TYPE ST_SafetyDoor_IN :
STRUCT
	bStartButton : BOOL;
	bRequestButton : BOOL;
	bLockButton : BOOL;
	bLocked : BOOL;
	tsSafe : BOOL;
	tsOpen : BOOL;
	tsSegment_Open : BOOL;
END_STRUCT
END_TYPE

(* stored: Version 1.1.0.1
   DUT ST_SafetyDoor_IN: Id {34f76f3d-388d-4cac-9a9e-326860192574} *)
